// LS Electric XG5000 project: 신호등
// PLC NewPLC

PROGRAM NewProgram (task: 스캔 프로그램)

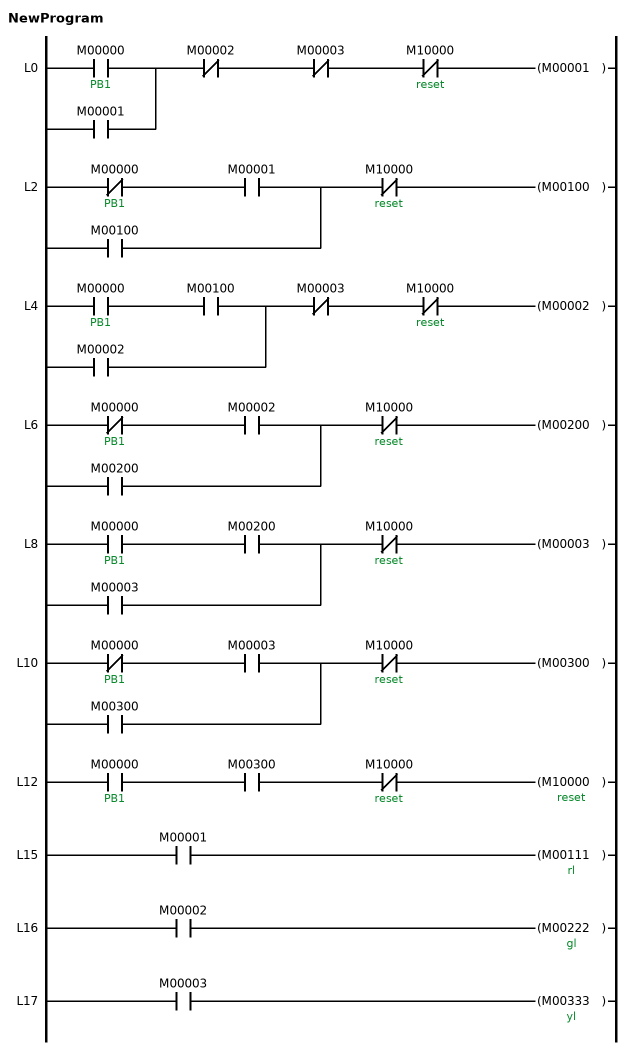
; L0
LOAD      M00000	// PB1
OR        M00001
AND NOT   M00002
AND NOT   M00003
AND NOT   M10000	// reset
OUT       M00001
; L2
LOAD NOT  M00000	// PB1
AND       M00001
OR        M00100
AND NOT   M10000	// reset
OUT       M00100
; L4
LOAD      M00000	// PB1
AND       M00100
OR        M00002
AND NOT   M00003
AND NOT   M10000	// reset
OUT       M00002
; L6
LOAD NOT  M00000	// PB1
AND       M00002
OR        M00200
AND NOT   M10000	// reset
OUT       M00200
; L8
LOAD      M00000	// PB1
AND       M00200
OR        M00003
AND NOT   M10000	// reset
OUT       M00003
; L10
LOAD NOT  M00000	// PB1
AND       M00003
OR        M00300
AND NOT   M10000	// reset
OUT       M00300
; L12
LOAD      M00000	// PB1
AND       M00300
AND NOT   M10000	// reset
OUT       M10000	// reset
; L15
LOAD      M00001
OUT       M00111	// rl
; L16
LOAD      M00002
OUT       M00222	// gl
; L17
LOAD      M00003
OUT       M00333	// yl